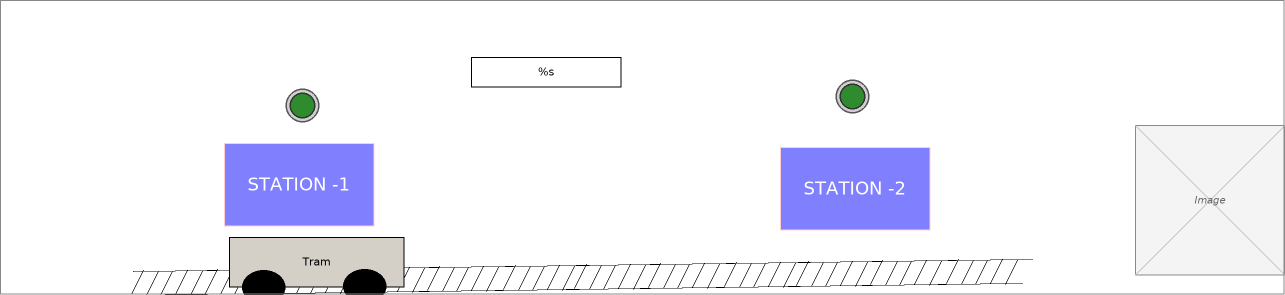
VISUALIZATION Visualization  // 1285x295
    Group (123,270 94x25)
        Line (0,25) (84,24)
        Line (20,0) (8,24)
        Line (35,1) (23,25)
        Line (49,1) (37,25)
        Line (64,0) (52,24)
        Line (79,1) (67,25)
        Line (10,1) (94,0)
    Group (197,269 94x25)
        Line (0,25) (84,24)
        Line (20,0) (8,24)
        Line (35,1) (23,25)
        Line (49,1) (37,25)
        Line (64,0) (52,24)
        Line (79,1) (67,25)
        Line (10,1) (94,0)
    Group (273,268 94x25)
        Line (0,25) (84,24)
        Line (20,0) (8,24)
        Line (35,1) (23,25)
        Line (49,1) (37,25)
        Line (64,0) (52,24)
        Line (79,1) (67,25)
        Line (10,1) (94,0)
    Group (345,267 94x25)
        Line (0,25) (84,24)
        Line (20,0) (8,24)
        Line (35,1) (23,25)
        Line (49,1) (37,25)
        Line (64,0) (52,24)
        Line (79,1) (67,25)
        Line (10,1) (94,0)
    Group (419,266 94x25)
        Line (0,25) (84,24)
        Line (20,0) (8,24)
        Line (35,1) (23,25)
        Line (49,1) (37,25)
        Line (64,0) (52,24)
        Line (79,1) (67,25)
        Line (10,1) (94,0)
    Group (495,265 94x25)
        Line (0,25) (84,24)
        Line (20,0) (8,24)
        Line (35,1) (23,25)
        Line (49,1) (37,25)
        Line (64,0) (52,24)
        Line (79,1) (67,25)
        Line (10,1) (94,0)
    Group (566,264 94x25)
        Line (0,25) (84,24)
        Line (20,0) (8,24)
        Line (35,1) (23,25)
        Line (49,1) (37,25)
        Line (64,0) (52,24)
        Line (79,1) (67,25)
        Line (10,1) (94,0)
    Group (640,263 94x25)
        Line (0,25) (84,24)
        Line (20,0) (8,24)
        Line (35,1) (23,25)
        Line (49,1) (37,25)
        Line (64,0) (52,24)
        Line (79,1) (67,25)
        Line (10,1) (94,0)
    Group (716,262 94x25)
        Line (0,25) (84,24)
        Line (20,0) (8,24)
        Line (35,1) (23,25)
        Line (49,1) (37,25)
        Line (64,0) (52,24)
        Line (79,1) (67,25)
        Line (10,1) (94,0)
    Group (788,261 94x25)
        Line (0,25) (84,24)
        Line (20,0) (8,24)
        Line (35,1) (23,25)
        Line (49,1) (37,25)
        Line (64,0) (52,24)
        Line (79,1) (67,25)
        Line (10,1) (94,0)
    Group (862,260 94x25)
        Line (0,25) (84,24)
        Line (20,0) (8,24)
        Line (35,1) (23,25)
        Line (49,1) (37,25)
        Line (64,0) (52,24)
        Line (79,1) (67,25)
        Line (10,1) (94,0)
    Group (938,259 94x25)
        Line (0,25) (84,24)
        Line (20,0) (8,24)
        Line (35,1) (23,25)
        Line (49,1) (37,25)
        Line (64,0) (52,24)
        Line (79,1) (67,25)
        Line (10,1) (94,0)
    Lamp1 (278,86 49x39), variable: GVL.qiAtStation1, style: Lamp-Lamp1-Green
    Lamp1 (828,77 49x39), variable: GVL.qiAtStation2, style: Lamp-Lamp1-Green
    Group (229,237 125x50)
        p3560616238: Process.Tramp_FB.AtPos
        RoundedRectangle (0,0 175x50), "Tram"
        Ellipse (13,33 43x34)
        Ellipse (114,32 43x34)
    Image (1135,125 150x150)
    RoundedRectangle (780,147 150x83), "STATION -2"
    RoundedRectangle (224,143 150x83), "STATION -1"
    Rectangle (471,57 150x30), "%s", text variable: GVL.qiDisplay
END_VISUALIZATION

(* stored: Version 1.1.0.1, ProductVersion 3.1.4024.12
   Visu Visualization: Id {9c57b31e-65a9-4b92-9580-d1593ceb7aae} *)
